FUNCTION_BLOCK bfb_fri_classifier
  (* Standard: 61499-2 *)
  (* Version 0.1, 2018-00-07, hpea485, UOA *)
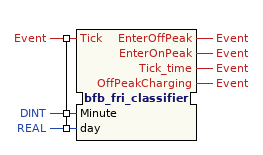
  EVENT_INPUT
    Tick WITH Minute, day;
  END_EVENT
  EVENT_OUTPUT
    EnterOffPeak;
    EnterOnPeak;
    Tick_time;
    OffPeakCharging;
  END_EVENT
  VAR_INPUT
    Minute : DINT;
    day : REAL;
  END_VAR
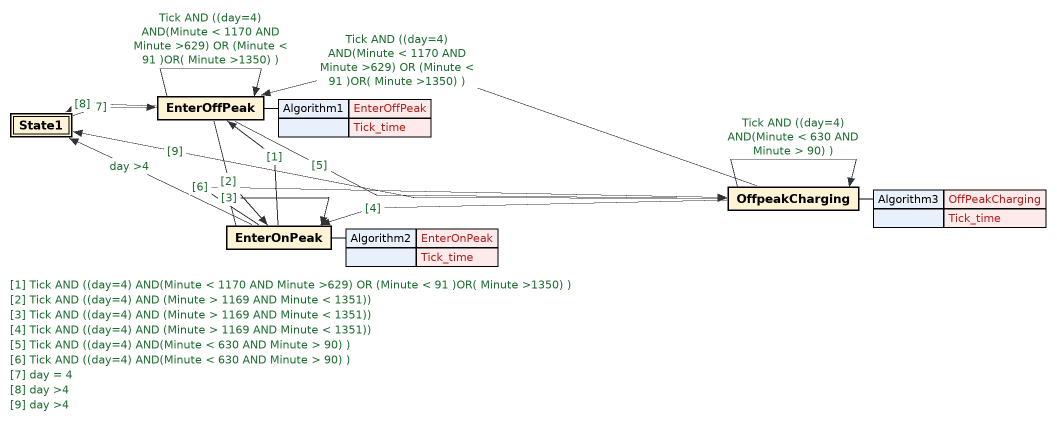
  EC_STATES
    State1;
    EnterOffPeak : Algorithm1 -> EnterOffPeak, -> Tick_time;
    EnterOnPeak : Algorithm2 -> EnterOnPeak, -> Tick_time;
    OffpeakCharging : Algorithm3 -> OffPeakCharging, -> Tick_time;
  END_STATES
  EC_TRANSITIONS
    EnterOffPeak TO EnterOffPeak := Tick AND ((day=4) AND(Minute < 1170 AND Minute >629) OR (Minute < 91 )OR( Minute >1350) );
    EnterOffPeak TO EnterOnPeak := Tick AND ((day=4) AND (Minute > 1169 AND Minute < 1351));
    EnterOffPeak TO OffpeakCharging := Tick AND ((day=4) AND(Minute < 630 AND Minute > 90) );
    EnterOffPeak TO State1 := day >4;
    EnterOnPeak TO EnterOnPeak := Tick AND ((day=4) AND (Minute > 1169 AND Minute < 1351));
    EnterOnPeak TO EnterOffPeak := Tick AND ((day=4) AND(Minute < 1170 AND Minute >629) OR (Minute < 91 )OR( Minute >1350) );
    EnterOnPeak TO OffpeakCharging := Tick AND ((day=4) AND(Minute < 630 AND Minute > 90) );
    EnterOnPeak TO State1 := day >4;
    OffpeakCharging TO OffpeakCharging := Tick AND ((day=4) AND(Minute < 630 AND Minute > 90) );
    OffpeakCharging TO EnterOnPeak := Tick AND ((day=4) AND (Minute > 1169 AND Minute < 1351));
    OffpeakCharging TO EnterOffPeak := Tick AND ((day=4) AND(Minute < 1170 AND Minute >629) OR (Minute < 91 )OR( Minute >1350) );
    OffpeakCharging TO State1 := day >4;
    State1 TO EnterOffPeak := day = 4;
  END_TRANSITIONS
  ALGORITHM Algorithm1 IN C:
printf("Entered OFF PEAK.....\r\n");
  END_ALGORITHM
  ALGORITHM Algorithm2 IN C:
printf(" Entered On peak .....\r\n ");
  END_ALGORITHM
  ALGORITHM Algorithm3 IN C:
printf(" OffPeak Charging \r\n ");
  END_ALGORITHM
END_FUNCTION_BLOCK
